FUNCTION_BLOCK Test_TEventHandler_HandlesRaisedEvent_UsingEventArgs EXTENDS T_UnitTestbase
VAR_INPUT
END_VAR
VAR_OUTPUT
END_VAR
VAR
    TestEvent : T_TestEvent_UsesEventArgs;
    TestEventHandler1 : T_TestEventHandler_UsesEventArgs;
    TestEventHandler2 : T_TestEventHandler_UsesEventArgs;
    TestEventHandler3 : T_TestEventHandler_UsesEventArgs;
    TestEventHandler4 : T_TestEventHandler_UsesEventArgs;
    TestEventHandler5 : T_TestEventHandler_UsesEventArgs;
END_VAR

TestEvent
    .ClearEventHandlers()
    .AddEventHandler(TestEventHandler1)
    .AddEventHandler(TestEventHandler2)
    .AddEventHandler(TestEventHandler3)
    .AddEventHandler(TestEventHandler4)
    .AddEventHandler(TestEventHandler5);
    
TestEvent.Args
    .Add_UDINT(21)
    .Add_LREAL(1.23)
    .Add_STRING('OnePointTwoThree')
    .Add_STRING('Big Long String')
    .Add_BOOL(TRUE);    
TestEvent.Raise();

Assertion.AssertEquals_BOOL(
    Expected := TRUE,
    Actual   := TestEventHandler1.EventWasRaised,
    VariableName  := 'TestEventHandler1.EventWasRaised');

Assertion.AssertEquals_BOOL(
    Expected := TRUE,
    Actual   := TestEventHandler2.EventWasRaised,
    VariableName  := 'TestEventHandler2.EventWasRaised');

Assertion.AssertEquals_BOOL(
    Expected := TRUE,
    Actual   := TestEventHandler3.EventWasRaised,
    VariableName  := 'TestEventHandler3.EventWasRaised');

Assertion.AssertEquals_BOOL(
    Expected := TRUE,
    Actual   := TestEventHandler4.EventWasRaised,
    VariableName  := 'TestEventHandler4.EventWasRaised');

Assertion.AssertEquals_BOOL(
    Expected := TRUE,
    Actual   := TestEventHandler5.EventWasRaised,
    VariableName  := 'TestEventHandler5.EventWasRaised');

    
Assertion.AssertEquals_UDINT(
    Expected := 21,
    Actual   := TestEventHandler1.Arg1,
    VariableName  := 'TestEventHandler1._EventData');
    
Assertion.AssertEquals_LREAL(
    Expected := 1.23,
    Actual   := TestEventHandler2.Arg2,
    Delta    := 0.000001,
    VariableName  := 'TestEventHandler2.Arg2');
    
Assertion.AssertEquals_STRING(
    Expected := 'OnePointTwoThree',
    Actual   := TestEventHandler3.Arg3,
    VariableName  := 'TestEventHandler3.Arg3');
    
Assertion.AssertEquals_STRING(
    Expected := 'Big Long String',
    Actual   := TestEventHandler4.Arg4,
    VariableName  := 'TestEventHandler4.Arg4');
    
Assertion.AssertEquals_BOOL(
    Expected := TRUE,
    Actual   := TestEventHandler5.Arg5,
    VariableName  := 'TestEventHandler5.Arg5');
    
TestFinished();

END_FUNCTION_BLOCK

(* stored: Version 1.1.0.1, ProductVersion 3.1.4024.4
   POU Test_TEventHandler_HandlesRaisedEvent_UsingEventArgs: Id {a335b2da-9644-416e-b62b-207f8baf078a}, SpecialFunc None *)
